// TIA Portal V19 export
DATA_BLOCK "A0301_Ribaltatore"   // DB77
// stored: InstanceOfName A0301_Ribaltatore_FB, InstanceOfType FB
"A0301_Ribaltatore_FB"
   // VAR_INPUT
   //    AreaInterface : "AreaInterface";
   //    ZSI : "udt_ZoneSafetyInterface";
   //    DSI_Feed : "udt_DeviceSafetyInterface";
   //    DSI_Valve : "udt_DeviceSafetyInterface";
   //    Drive : "TAx_DriveInterface";
   //    DataIn : Struct
   //       OP_MoveToPos_PB : Bool;
   //       OP_Rest_PB : Bool;
   //       OP_Work_PB : Bool;
   //    END_STRUCT;
   //    CIn { ExternalAccessible := 'False'; ExternalVisible := 'False'; ExternalWritable := 'False'} : Struct
   //       Manager : Struct
   //          Ax : "Positioning_EPOS_Machine_Manager";
   //          Solleva : "ValveMachine_Manager";
   //       END_STRUCT;
   //       SemiAut_PB : Bool;
   //       Ax_Req : Struct
   //          Pos0 : Bool;
   //          Pos1 : Bool;
   //          Pos2 : Bool;
   //          Pos3 : Bool;
   //       END_STRUCT;
   //       P2 : Struct
   //          Fermi : "ValveMachine_COut";
   //          Sollevatore : "ValveMachine_COut";
   //       END_STRUCT;
   //       P3 : Struct
   //          Fermi : "ValveMachine_COut";
   //       END_STRUCT;
   //       P4 : Struct
   //          Fermi : "ValveMachine_COut";
   //       END_STRUCT;
   //       Trasporto : "SpeedMachine_COut";
   //    END_STRUCT;
   //    Config : Struct
   //       Ax : "Positioning_EPOS_Machine_Config_NEW";
   //       Solleva_Rib : Array[1..6] of "ValveMachine_Config";
   //    END_STRUCT;
   //    HWID_Ax_TEL111 : HW_SUBMODULE;
   // END_VAR
   // VAR_OUTPUT
   //    MachineInterface { ExternalAccessible := 'False'; ExternalVisible := 'False'; ExternalWritable := 'False'} : "MachineInterface";
   //    DataOut : "Positioning_EPOS_Machine_DataOut";
   //    COut : Struct
   //       Solleva_Rib : "ValveMachine_COut";
   //       Ribaltatore : "Positioning_EPOS_Machine_COut";
   //       Ribaltatore_Sts : Struct
   //          Pos0_Reached : Bool;
   //          Pos1_Reached : Bool;
   //          Pos2_Reached : Bool;
   //          Pos3_Reached : Bool;
   //       END_STRUCT;
   //       Ribaltatore_AtRest : Bool;
   //    END_STRUCT;
   // END_VAR
   // VAR_IN_OUT
   //    Par_Manu : "Positioning_EPOS_Machine_Par";
   //    Par_Aut : "A0301_Mach_Ribaltatore_Par";
   //    Pers_Data : Struct
   //       EncoderAbsolute_Preset_OK : Bool;
   //       Persistent_ActualPosition : LReal;
   //    END_STRUCT;
   // END_VAR
   // VAR
   //    Alarm : Struct
   //       Solleva_Rib { S7_SetPoint := 'True'} : Array[1..6] of "ValveAlr";
   //       Ax { ExternalVisible := 'False'} : "Positioning_EPOS_Machine_Alr";
   //    END_STRUCT;
   //    Warning : Struct
   //       Ax { S7_SetPoint := 'True'} : "Positioning_EPOS_Machine_Wng";
   //       Solleva_Rib { S7_SetPoint := 'True'} : Array[1..6] of "ValveMachine_Wng";
   //       OP_REST_MissingCnd : Bool;
   //       OP_WORK_MissingCnd : Bool;
   //    END_STRUCT;
   //    ValueVelOvr { ExternalAccessible := 'False'; ExternalVisible := 'False'; ExternalWritable := 'False'} : Array[1..10] of Real;
   //    Ax : "Positioning_EPOS_Machine_FB_NEW";
   //    Solleva_Rib { S7_SetPoint := 'True'} : Array[1..6] of "ValveMachine_FB";
   //    TON : Struct
   //       DelayPos1_SG : IEC_TIMER;
   //    END_STRUCT;
   //    Sts : Struct
   //       ReadyForMove : Bool;
   //       OP_CanMoveFreely : Bool;
   //       OP_MoveToPos_Cnd : Bool;
   //       OP_Rest_Cnd : Bool;
   //       OP_Work_Cnd : Bool;
   //       Solleva_Rib_AlarmPresence : Bool;
   //    END_STRUCT;
   //    Ctrl : Struct
   //       Ribaltatore : Struct
   //          OP_MoveToPos : Bool;
   //          Ax_MoveToPos : Bool;
   //       END_STRUCT;
   //       Solleva : Struct
   //          OP_Rest_Man : Bool;
   //          OP_Work_Man : Bool;
   //          OP_Rest_Aut : Bool;
   //          OP_Work_Aut : Bool;
   //          OP_Rest : Bool;
   //          OP_Work : Bool;
   //       END_STRUCT;
   //    END_STRUCT;
   //    HMI : Struct
   //       Ax : Struct
   //          B_Preset : Bool;
   //          PresetPosition : LReal;
   //          TargetPosition : LReal;
   //       END_STRUCT;
   //       SollevaRibSts { S7_SetPoint := 'True'} : "UDT_HMI-Sts_ValvePosA0301";
   //       OP_Sel_Pos0 : Bool;
   //       OP_Sel_Pos1 : Bool;
   //       OP_Sel_Pos2 : Bool;
   //       OP_Sel_Pos3 : Bool;
   //    END_STRUCT;
   //    AUX : Struct
   //       Solleva_Rib : Struct
   //          OP_Rest_PB : Bool;
   //          OP_Work_PB : Bool;
   //       END_STRUCT;
   //       Ribaltatore : Struct
   //          Ax_MoveToPos_PB : Bool;
   //       END_STRUCT;
   //    END_STRUCT;
   //    TON_Anticipi : Struct
   //       Rest : Struct
   //          SollevaRib { S7_SetPoint := 'True'} : IEC_TIMER;
   //       END_STRUCT;
   //       Work : Struct
   //          SollevaRib : IEC_TIMER;
   //       END_STRUCT;
   //    END_STRUCT;
   // END_VAR
BEGIN
END_DATA_BLOCK
